FUNCTION Convert_TIME_TO_STRING : BOOL
VAR_INPUT
	in : TIME;
	out : REFERENCE TO STRING;
END_VAR
VAR
	converted : STRING;
END_VAR

converted := TIME_TO_STRING(in);

IF (STRING_TO_TIME(converted) <> in) THEN
	RETURN;
END_IF

out := converted;
Convert_TIME_TO_STRING := TRUE;

END_FUNCTION

(* stored: Version 1.1.0.1, ProductVersion 3.1.4024.12
   POU Convert_TIME_TO_STRING: Id {a082cc42-2f97-44e7-a7cd-ac925f4b6ff7}, SpecialFunc None *)
